TYPE ST_SA :
STRUCT
	name		: STRING;
	ID			: INT;
	EstopOK		: BOOL;
	GatesOK		: BOOL;
	SafetyOK	: BOOL;
END_STRUCT
END_TYPE

(* stored: Version 1.1.0.1
   DUT ST_SA: Id {e0a2e851-3760-433e-9f36-0f7c493cd5f8} *)
